{attribute 'linkalways'} 
{attribute 'no_explicit_call' := 'This FB is a CLASS and must be accessed using methods or properties'}
{attribute 'enable_dynamic_creation'}
FUNCTION_BLOCK FINAL LT_USINT EXTENDS Node
VAR
	in1 : _USINT(0);
	in2 : _USINT(0);
	out : _BOOL(FALSE);
END_VAR

METHOD PUBLIC Clone : I_Node
VAR
	pNode : POINTER TO LT_USINT;
END_VAR
pNode := __NEW(LT_USINT);
Clone := pNode^;
END_METHOD

METHOD FB_init : BOOL
VAR_INPUT
	bInitRetains : BOOL; // if TRUE, the retain variables are initialized (warm start / cold start)
	bInCopyCode : BOOL;  // if TRUE, the instance afterwards gets moved into the copy code (online change)
END_VAR
AddInput('in1',THIS^.in1);
AddInput('in2',THIS^.in2);
AddOutput('out', THIS^.out);
END_METHOD

METHOD PROTECTED OnExecute
VAR
END_VAR
out.Value := in1.Value < in2.Value;
END_METHOD

END_FUNCTION_BLOCK

(* stored: Version 1.1.0.1, ProductVersion 3.1.4024.15
   POU LT_USINT: Id {e20da5a9-70bb-4539-b71b-fad38c72033b}, SpecialFunc None
   Folder Constructor: Id {6b121032-184a-4ced-9c09-ad26fa772b7a}
   Method Clone: Id {5c53d8c1-fbc9-4ebe-8f21-d9706b9b2ade}
   Method FB_init: Id {380b9a6e-83be-4a67-b2c5-6ee5b9b6d456}
   Method OnExecute: Id {1f0606cd-ab07-49ae-9666-1cdb6c5086d2} *)
